{attribute 'qualified_only'}
{attribute 'strict'}
{attribute 'to_string'}

TYPE E_Request :
(
	{attribute 'hide'}
    Undefined   := 0,
	{attribute 'analysis' := '-27'}
	Reset       := 1,
	{attribute 'analysis' := '-27'}
    Start       := 2,
	{attribute 'analysis' := '-27'}
	Complete	:= 3,
	{attribute 'analysis' := '-27'}
	Stop		:= 4,
	{attribute 'analysis' := '-27'}
	Abort		:= 8
);
END_TYPE

(* stored: Version 1.1.0.1
   DUT E_Request: Id {d3b20770-b5da-468b-8276-148bae048ad0} *)
